// TIA Portal V20 export
DATA_BLOCK "FB_IO_Map_Disp_IDB"   // DB101
// stored: AutoNumber false, InstanceOfName FB_IO_Map_Disp, InstanceOfType FB
"FB_IO_Map_Disp"
   // VAR
   //    Start_Address_IByte : UInt;
   //    Start_Address_OByte : UInt;
   //    Start_Address_SIByte : UDInt := 30000;
   //    Start_Address_SOByte : UDInt := 31000;
   //    Loop_I : Int;
   //    Input : Array[0..15] of Bool;
   //    SInput : Array[0..15] of Bool;
   //    Loop_O : Int;
   //    Output : Array[0..15] of Bool;
   //    SOutput : Array[0..15] of Bool;
   // END_VAR
BEGIN
END_DATA_BLOCK
